{attribute 'enable_dynamic_creation'}
TYPE Node :
STRUCT
	data : INT;
	next : POINTER TO Node;
END_STRUCT
END_TYPE

(* stored: Version 1.1.0.1, ProductVersion 3.1.4024.9
   DUT Node: Id {ec13c4f1-266e-482d-9b20-9541e4253173} *)
